FUNCTION FC_ToByte : BOOL
VAR_INPUT
	RegSource : POINTER TO BOOL;
	RegDest	  : POINTER TO BYTE;
	Size : UINT;
END_VAR
VAR
	i 	: DINT;
	j   : DINT;
	bitIndex : INT;
	byteIndex : INT;
	temp : BYTE;
END_VAR

FOR i:=0 TO size-1 BY 8 DO
	temp := 0;
	FOR j:= 0 TO 7 DO
		IF RegSource[i+j] THEN
			temp := temp OR (SHL(1,j));
		END_IF
	END_FOR
	RegDest^ := temp;
	RegDest:=RegDest+1;
END_FOR

END_FUNCTION

(* stored: Version 1.1.0.1, ProductVersion 3.1.4024.13
   POU FC_ToByte: Id {e061983b-0fff-427f-aace-29ee9eeee981}, SpecialFunc None *)
